// TIA Portal V17 export
// export: Created 2022-07-20T06:59:49.090747Z, ExportSetting WithDefaults, DisplayName Totally Integrated Automation Portal, DisplayVersion V17, DisplayName TIA Portal Openness, DisplayVersion V17, DisplayName TIA Portal Version Control Interface, DisplayVersion V17, DisplayName SINAMICS Startdrive Advanced, DisplayVersion V17, DisplayName SINAMICS Startdrive G130, G150, S120, S150, SINAMICS MV, S210, DisplayVersion V17, DisplayName SINAMICS Startdrive G110M, G120, G120C, G120D, G120P, G115D, DisplayVersion V17, DisplayName STEP 7 Professional, DisplayVersion V17, DisplayName STEP 7 Safety, DisplayVersion V17, DisplayName WinCC Advanced, DisplayVersion V17
FUNCTION_BLOCK "FB10220_OperatingTimeCounter"   // FB10220, LAD
TITLE = FB10220_OperatingTimeCounter
{ S7_Optimized_Access := 'TRUE' }
AUTHOR : Anirouddh
FAMILY : 1022x_COUNTERS
VERSION : 1.0
// Release note : 
// 1.0 - Feature developped
// stored: AutoNumber false, IsIECCheckEnabled false, IsRetainMemResEnabled false, MemoryReserve 100, SetENOAutomatically false, UDAEnableTagReadback false
   VAR_INPUT
      SignalToCount : Bool;
   END_VAR
   VAR_IN_OUT
      ResetCounter : Bool;
      ElapsedTime : LReal;   // in s
   END_VAR
   VAR
      R_TRIG_Clock_100ms { S7_SetPoint := 'True'} : R_TRIG;
   END_VAR
BEGIN

REGION Network 1 (SCL): Edge Signals & Timers Management
   REGION EDGE SIGNALS
       #R_TRIG_Clock_100ms(CLK := "Clock_10Hz");
   END_REGION
END_REGION

REGION Network 2 (SCL): Time Counter Management
   IF #SignalToCount AND #R_TRIG_Clock_100ms.Q THEN
       #ElapsedTime += 0.1;
   ELSIF #ResetCounter THEN
       #ElapsedTime := 0.0;
       IF #ElapsedTime = 0.0 THEN
           #ResetCounter := FALSE;
       END_IF;
   END_IF;
END_REGION
END_FUNCTION_BLOCK
